    movel([0.601016, -1.382739, -2.575796, -0.753854, 1.570796, 2.171812],accel_mss,speed_ms,0,blend_radius_m)
    movel([0.599309, -1.384316, -2.574679, -0.753394, 1.570796, 2.170106],accel_mss,speed_ms,0,blend_radius_m)
    movel([0.597574, -1.385721, -2.573681, -0.752987, 1.570796, 2.168370],accel_mss,speed_ms,0,blend_radius_m)
    movel([0.595833, -1.386908, -2.572835, -0.752646, 1.570796, 2.166630],accel_mss,speed_ms,0,blend_radius_m)
    movel([0.594095, -1.387836, -2.572173, -0.752380, 1.570796, 2.164892],accel_mss,speed_ms,0,blend_radius_m)
    movel([0.592375, -1.388464, -2.571724, -0.752201, 1.570796, 2.163171],accel_mss,speed_ms,0,blend_radius_m)
    movel([0.590691, -1.388744, -2.571523, -0.752121, 1.570796, 2.161487],accel_mss,speed_ms,0,blend_radius_m)
    movel([0.589052, -1.388638, -2.571599, -0.752152, 1.570796, 2.159848],accel_mss,speed_ms,0,blend_radius_m)
    movel([0.588253, -1.388424, -2.571753, -0.752213, 1.570796, 2.159050],accel_mss,speed_ms,0,blend_radius_m)
    movel([0.587471, -1.388096, -2.571987, -0.752306, 1.570796, 2.158268],accel_mss,speed_ms,0,blend_radius_m)
    movel([0.585965, -1.387077, -2.572715, -0.752597, 1.570796, 2.156761],accel_mss,speed_ms,0,blend_radius_m)
    movel([0.584424, -1.385537, -2.573812, -0.753040, 1.570796, 2.155220],accel_mss,speed_ms,0,blend_radius_m)
    movel([0.583153, -1.383849, -2.575010, -0.753530, 1.570796, 2.153949],accel_mss,speed_ms,0,blend_radius_m)
    movel([0.582122, -1.382027, -2.576299, -0.754063, 1.570796, 2.152918],accel_mss,speed_ms,0,blend_radius_m)
    movel([0.581300, -1.380074, -2.577675, -0.754640, 1.570796, 2.152096],accel_mss,speed_ms,0,blend_radius_m)
    movel([0.580659, -1.378000, -2.579131, -0.755258, 1.570796, 2.151455],accel_mss,speed_ms,0,blend_radius_m)
    movel([0.580165, -1.375815, -2.580658, -0.755917, 1.570796, 2.150961],accel_mss,speed_ms,0,blend_radius_m)
    movel([0.579497, -1.371134, -2.583905, -0.757350, 1.570796, 2.150294],accel_mss,speed_ms,0,blend_radius_m)
    movel([0.578951, -1.365850, -2.587534, -0.759005, 1.570796, 2.149747],accel_mss,speed_ms,0,blend_radius_m)
    movel([0.578551, -1.360508, -2.591161, -0.760719, 1.570796, 2.149347],accel_mss,speed_ms,0,blend_radius_m)
    movel([0.578456, -1.355007, -2.594855, -0.762526, 1.570796, 2.149252],accel_mss,speed_ms,0,blend_radius_m)
    movel([0.578578, -1.352162, -2.596749, -0.763478, 1.570796, 2.149375],accel_mss,speed_ms,0,blend_radius_m)
    movel([0.578843, -1.349233, -2.598687, -0.764469, 1.570796, 2.149640],accel_mss,speed_ms,0,blend_radius_m)
    movel([0.579128, -1.345588, -2.601082, -0.765719, 1.570796, 2.149924],accel_mss,speed_ms,0,blend_radius_m)
    movel([0.579166, -1.341949, -2.603455, -0.766985, 1.570796, 2.149962],accel_mss,speed_ms,0,blend_radius_m)
    movel([0.578983, -1.338332, -2.605795, -0.768262, 1.570796, 2.149780],accel_mss,speed_ms,0,blend_radius_m)
    movel([0.578620, -1.334746, -2.608097, -0.769545, 1.570796, 2.149417],accel_mss,speed_ms,0,blend_radius_m)
    movel([0.577474, -1.327732, -2.612550, -0.772107, 1.570796, 2.148271],accel_mss,speed_ms,0,blend_radius_m)
    movel([0.576003, -1.321005, -2.616758, -0.774626, 1.570796, 2.146800],accel_mss,speed_ms,0,blend_radius_m)
    movel([0.574612, -1.316084, -2.619798, -0.776507, 1.570796, 2.145408],accel_mss,speed_ms,0,blend_radius_m)
    movel([0.572792, -1.311386, -2.622670, -0.778332, 1.570796, 2.143588],accel_mss,speed_ms,0,blend_radius_m)
    movel([0.570532, -1.306949, -2.625357, -0.780084, 1.570796, 2.141328],accel_mss,speed_ms,0,blend_radius_m)
    movel([0.567821, -1.302820, -2.627833, -0.781736, 1.570796, 2.138617],accel_mss,speed_ms,0,blend_radius_m)
    movel([0.564652, -1.299032, -2.630085, -0.783272, 1.570796, 2.135448],accel_mss,speed_ms,0,blend_radius_m)
    movel([0.562893, -1.297282, -2.631119, -0.783988, 1.570796, 2.133689],accel_mss,speed_ms,0,blend_radius_m)
    movel([0.559022, -1.294091, -2.632994, -0.785303, 1.570796, 2.129818],accel_mss,speed_ms,0,blend_radius_m)
    movel([0.556907, -1.292661, -2.633831, -0.785897, 1.570796, 2.127704],accel_mss,speed_ms,0,blend_radius_m)
    movel([0.552322, -1.290161, -2.635286, -0.786941, 1.570796, 2.123118],accel_mss,speed_ms,0,blend_radius_m)
    movel([0.548890, -1.288814, -2.636068, -0.787508, 1.570796, 2.119686],accel_mss,speed_ms,0,blend_radius_m)
    movel([0.545173, -1.287852, -2.636624, -0.787913, 1.570796, 2.115969],accel_mss,speed_ms,0,blend_radius_m)
    movel([0.541202, -1.287290, -2.636948, -0.788150, 1.570796, 2.111998],accel_mss,speed_ms,0,blend_radius_m)
    movel([0.537005, -1.287149, -2.637030, -0.788210, 1.570796, 2.107801],accel_mss,speed_ms,0,blend_radius_m)
    movel([0.532609, -1.287443, -2.636860, -0.788086, 1.570796, 2.103406],accel_mss,speed_ms,0,blend_radius_m)
    movel([0.528049, -1.288183, -2.636433, -0.787773, 1.570796, 2.098845],accel_mss,speed_ms,0,blend_radius_m)
    movel([0.523356, -1.289383, -2.635738, -0.787268, 1.570796, 2.094152],accel_mss,speed_ms,0,blend_radius_m)
    movel([0.518564, -1.291050, -2.634770, -0.786569, 1.570796, 2.089360],accel_mss,speed_ms,0,blend_radius_m)
    movel([0.514066, -1.292974, -2.633648, -0.785767, 1.570796, 2.084862],accel_mss,speed_ms,0,blend_radius_m)
    movel([0.509727, -1.295149, -2.632374, -0.784866, 1.570796, 2.080523],accel_mss,speed_ms,0,blend_radius_m)
    movel([0.505563, -1.297588, -2.630938, -0.783862, 1.570796, 2.076360],accel_mss,speed_ms,0,blend_radius_m)
    movel([0.501589, -1.300304, -2.629331, -0.782754, 1.570796, 2.072386],accel_mss,speed_ms,0,blend_radius_m)
    movel([0.499677, -1.301770, -2.628459, -0.782160, 1.570796, 2.070473],accel_mss,speed_ms,0,blend_radius_m)
    movel([0.496018, -1.304922, -2.626575, -0.780892, 1.570796, 2.066815],accel_mss,speed_ms,0,blend_radius_m)
    movel([0.494274, -1.306613, -2.625559, -0.780217, 1.570796, 2.065071],accel_mss,speed_ms,0,blend_radius_m)
    movel([0.490969, -1.310226, -2.623376, -0.778788, 1.570796, 2.061765],accel_mss,speed_ms,0,blend_radius_m)
    movel([0.489409, -1.312153, -2.622204, -0.778032, 1.570796, 2.060205],accel_mss,speed_ms,0,blend_radius_m)
    movel([0.487917, -1.314158, -2.620980, -0.777252, 1.570796, 2.058713],accel_mss,speed_ms,0,blend_radius_m)
    movel([0.485915, -1.317093, -2.619178, -0.776118, 1.570796, 2.056711],accel_mss,speed_ms,0,blend_radius_m)
    movel([0.484053, -1.320085, -2.617329, -0.774975, 1.570796, 2.054849],accel_mss,speed_ms,0,blend_radius_m)
    movel([0.482333, -1.323108, -2.615449, -0.773832, 1.570796, 2.053129],accel_mss,speed_ms,0,blend_radius_m)
    movel([0.480751, -1.326147, -2.613547, -0.772695, 1.570796, 2.051547],accel_mss,speed_ms,0,blend_radius_m)
    movel([0.479315, -1.329177, -2.611638, -0.771574, 1.570796, 2.050111],accel_mss,speed_ms,0,blend_radius_m)
    movel([0.478026, -1.332177, -2.609736, -0.770476, 1.570796, 2.048823],accel_mss,speed_ms,0,blend_radius_m)
    movel([0.476884, -1.335130, -2.607852, -0.769407, 1.570796, 2.047680],accel_mss,speed_ms,0,blend_radius_m)
    movel([0.475891, -1.338015, -2.605999, -0.768375, 1.570796, 2.046688],accel_mss,speed_ms,0,blend_radius_m)
    movel([0.472966, -1.349149, -2.598742, -0.764497, 1.570796, 2.043762],accel_mss,speed_ms,0,blend_radius_m)
    movel([0.470619, -1.357979, -2.592865, -0.761545, 1.570796, 2.041416],accel_mss,speed_ms,0,blend_radius_m)
    movel([0.470325, -1.358818, -2.592301, -0.761270, 1.570796, 2.041122],accel_mss,speed_ms,0,blend_radius_m)
    movel([0.475631, -1.356833, -2.593634, -0.761922, 1.570796, 2.046427],accel_mss,speed_ms,0,blend_radius_m)
    movel([0.480943, -1.355196, -2.594729, -0.762464, 1.570796, 2.051739],accel_mss,speed_ms,0,blend_radius_m)
    movel([0.486236, -1.353899, -2.595594, -0.762896, 1.570796, 2.057033],accel_mss,speed_ms,0,blend_radius_m)
    movel([0.491479, -1.352929, -2.596240, -0.763220, 1.570796, 2.062275],accel_mss,speed_ms,0,blend_radius_m)
    movel([0.496639, -1.352279, -2.596672, -0.763438, 1.570796, 2.067435],accel_mss,speed_ms,0,blend_radius_m)
    movel([0.501690, -1.351932, -2.596902, -0.763555, 1.570796, 2.072486],accel_mss,speed_ms,0,blend_radius_m)
    movel([0.506601, -1.351881, -2.596936, -0.763573, 1.570796, 2.077398],accel_mss,speed_ms,0,blend_radius_m)
    movel([0.511345, -1.352106, -2.596786, -0.763497, 1.570796, 2.082141],accel_mss,speed_ms,0,blend_radius_m)
    movel([0.513503, -1.352345, -2.596628, -0.763416, 1.570796, 2.084300],accel_mss,speed_ms,0,blend_radius_m)
    movel([0.515622, -1.352729, -2.596373, -0.763287, 1.570796, 2.086418],accel_mss,speed_ms,0,blend_radius_m)
    movel([0.517679, -1.353257, -2.596022, -0.763110, 1.570796, 2.088475],accel_mss,speed_ms,0,blend_radius_m)
    movel([0.519651, -1.353929, -2.595574, -0.762885, 1.570796, 2.090447],accel_mss,speed_ms,0,blend_radius_m)
    movel([0.521517, -1.354747, -2.595029, -0.762613, 1.570796, 2.092314],accel_mss,speed_ms,0,blend_radius_m)
    movel([0.523257, -1.355711, -2.594385, -0.762293, 1.570796, 2.094053],accel_mss,speed_ms,0,blend_radius_m)
    movel([0.524849, -1.356818, -2.593644, -0.761927, 1.570796, 2.095645],accel_mss,speed_ms,0,blend_radius_m)
    movel([0.526273, -1.358067, -2.592806, -0.761516, 1.570796, 2.097069],accel_mss,speed_ms,0,blend_radius_m)
    movel([0.527508, -1.359460, -2.591868, -0.761060, 1.570796, 2.098304],accel_mss,speed_ms,0,blend_radius_m)
    movel([0.528536, -1.360996, -2.590832, -0.760561, 1.570796, 2.099332],accel_mss,speed_ms,0,blend_radius_m)
    movel([0.529334, -1.362671, -2.589697, -0.760020, 1.570796, 2.100130],accel_mss,speed_ms,0,blend_radius_m)
    movel([0.529883, -1.364486, -2.588464, -0.759439, 1.570796, 2.100680],accel_mss,speed_ms,0,blend_radius_m)
    movel([0.530165, -1.366437, -2.587133, -0.758820, 1.570796, 2.100962],accel_mss,speed_ms,0,blend_radius_m)
    movel([0.530163, -1.368526, -2.585701, -0.758162, 1.570796, 2.100960],accel_mss,speed_ms,0,blend_radius_m)
    movel([0.529857, -1.370747, -2.584172, -0.757470, 1.570796, 2.100654],accel_mss,speed_ms,0,blend_radius_m)
    movel([0.529228, -1.373102, -2.582544, -0.756743, 1.570796, 2.100024],accel_mss,speed_ms,0,blend_radius_m)
    movel([0.528005, -1.376258, -2.580348, -0.755782, 1.570796, 2.098801],accel_mss,speed_ms,0,blend_radius_m)
    movel([0.526428, -1.379471, -2.578099, -0.754819, 1.570796, 2.097224],accel_mss,speed_ms,0,blend_radius_m)
    movel([0.524564, -1.382702, -2.575822, -0.753865, 1.570796, 2.095360],accel_mss,speed_ms,0,blend_radius_m)
    movel([0.522477, -1.385922, -2.573537, -0.752929, 1.570796, 2.093273],accel_mss,speed_ms,0,blend_radius_m)
    movel([0.520232, -1.389098, -2.571270, -0.752021, 1.570796, 2.091028],accel_mss,speed_ms,0,blend_radius_m)
    movel([0.517887, -1.392198, -2.569042, -0.751149, 1.570796, 2.088683],accel_mss,speed_ms,0,blend_radius_m)
    movel([0.513159, -1.398048, -2.564800, -0.749541, 1.570796, 2.083955],accel_mss,speed_ms,0,blend_radius_m)
    movel([0.510054, -1.401623, -2.562183, -0.748583, 1.570796, 2.080850],accel_mss,speed_ms,0,blend_radius_m)
    movel([0.506857, -1.405036, -2.559666, -0.747687, 1.570796, 2.077653],accel_mss,speed_ms,0,blend_radius_m)
    movel([0.503577, -1.408310, -2.557236, -0.746843, 1.570796, 2.074373],accel_mss,speed_ms,0,blend_radius_m)
    movel([0.500217, -1.411476, -2.554871, -0.746042, 1.570796, 2.071013],accel_mss,speed_ms,0,blend_radius_m)
    movel([0.496786, -1.414553, -2.552558, -0.745278, 1.570796, 2.067583],accel_mss,speed_ms,0,blend_radius_m)
    movel([0.493292, -1.417568, -2.550278, -0.744543, 1.570796, 2.064088],accel_mss,speed_ms,0,blend_radius_m)
    movel([0.486129, -1.423508, -2.545746, -0.743135, 1.570796, 2.056925],accel_mss,speed_ms,0,blend_radius_m)
    movel([0.487951, -1.426525, -2.543424, -0.742440, 1.570796, 2.058747],accel_mss,speed_ms,0,blend_radius_m)
    movel([0.488812, -1.428211, -2.542120, -0.742058, 1.570796, 2.059609],accel_mss,speed_ms,0,blend_radius_m)
    movel([0.489370, -1.429952, -2.540769, -0.741667, 1.570796, 2.060166],accel_mss,speed_ms,0,blend_radius_m)
    movel([0.489470, -1.430830, -2.540087, -0.741472, 1.570796, 2.060266],accel_mss,speed_ms,0,blend_radius_m)
    movel([0.489417, -1.431705, -2.539405, -0.741279, 1.570796, 2.060213],accel_mss,speed_ms,0,blend_radius_m)
    movel([0.489187, -1.432571, -2.538729, -0.741089, 1.570796, 2.059983],accel_mss,speed_ms,0,blend_radius_m)
    movel([0.488755, -1.433422, -2.538064, -0.740904, 1.570796, 2.059551],accel_mss,speed_ms,0,blend_radius_m)
    movel([0.488098, -1.434250, -2.537415, -0.740724, 1.570796, 2.058895],accel_mss,speed_ms,0,blend_radius_m)
    movel([0.487186, -1.435055, -2.536784, -0.740550, 1.570796, 2.057983],accel_mss,speed_ms,0,blend_radius_m)
    movel([0.485997, -1.435830, -2.536175, -0.740384, 1.570796, 2.056793],accel_mss,speed_ms,0,blend_radius_m)
    movel([0.484506, -1.436568, -2.535594, -0.740227, 1.570796, 2.055302],accel_mss,speed_ms,0,blend_radius_m)
    movel([0.483220, -1.437075, -2.535195, -0.740119, 1.570796, 2.054016],accel_mss,speed_ms,0,blend_radius_m)
    movel([0.482001, -1.437448, -2.534901, -0.740040, 1.570796, 2.052798],accel_mss,speed_ms,0,blend_radius_m)
    movel([0.480845, -1.437700, -2.534702, -0.739987, 1.570796, 2.051642],accel_mss,speed_ms,0,blend_radius_m)
    movel([0.478697, -1.437878, -2.534562, -0.739949, 1.570796, 2.049493],accel_mss,speed_ms,0,blend_radius_m)
    movel([0.477695, -1.437824, -2.534604, -0.739961, 1.570796, 2.048491],accel_mss,speed_ms,0,blend_radius_m)
    movel([0.475806, -1.437485, -2.534871, -0.740032, 1.570796, 2.046602],accel_mss,speed_ms,0,blend_radius_m)
    movel([0.474040, -1.436905, -2.535329, -0.740155, 1.570796, 2.044837],accel_mss,speed_ms,0,blend_radius_m)
    movel([0.472356, -1.436162, -2.535914, -0.740313, 1.570796, 2.043153],accel_mss,speed_ms,0,blend_radius_m)
    movel([0.469076, -1.434521, -2.537203, -0.740665, 1.570796, 2.039872],accel_mss,speed_ms,0,blend_radius_m)
    movel([0.465722, -1.436483, -2.535661, -0.740245, 1.570796, 2.036518],accel_mss,speed_ms,0,blend_radius_m)
    movel([0.463980, -1.437385, -2.534950, -0.740053, 1.570796, 2.034776],accel_mss,speed_ms,0,blend_radius_m)
    movel([0.462220, -1.438181, -2.534322, -0.739885, 1.570796, 2.033016],accel_mss,speed_ms,0,blend_radius_m)
    movel([0.460464, -1.438828, -2.533812, -0.739750, 1.570796, 2.031260],accel_mss,speed_ms,0,blend_radius_m)
    movel([0.458733, -1.439284, -2.533451, -0.739654, 1.570796, 2.029530],accel_mss,speed_ms,0,blend_radius_m)
    movel([0.457049, -1.439507, -2.533274, -0.739608, 1.570796, 2.027846],accel_mss,speed_ms,0,blend_radius_m)
    movel([0.455428, -1.439456, -2.533315, -0.739619, 1.570796, 2.026225],accel_mss,speed_ms,0,blend_radius_m)
    movel([0.454430, -1.439177, -2.533536, -0.739677, 1.570796, 2.025226],accel_mss,speed_ms,0,blend_radius_m)
    movel([0.453802, -1.438678, -2.533930, -0.739781, 1.570796, 2.024598],accel_mss,speed_ms,0,blend_radius_m)
    movel([0.453497, -1.437998, -2.534467, -0.739924, 1.570796, 2.024293],accel_mss,speed_ms,0,blend_radius_m)
    movel([0.453470, -1.437176, -2.535115, -0.740098, 1.570796, 2.024266],accel_mss,speed_ms,0,blend_radius_m)
    movel([0.453674, -1.436249, -2.535845, -0.740295, 1.570796, 2.024470],accel_mss,speed_ms,0,blend_radius_m)
    movel([0.454060, -1.435263, -2.536620, -0.740506, 1.570796, 2.024857],accel_mss,speed_ms,0,blend_radius_m)
    movel([0.454581, -1.434254, -2.537412, -0.740723, 1.570796, 2.025378],accel_mss,speed_ms,0,blend_radius_m)
    movel([0.455194, -1.433264, -2.538187, -0.740938, 1.570796, 2.025991],accel_mss,speed_ms,0,blend_radius_m)
    movel([0.456666, -1.431232, -2.539773, -0.741384, 1.570796, 2.027463],accel_mss,speed_ms,0,blend_radius_m)
    movel([0.458291, -1.429284, -2.541288, -0.741817, 1.570796, 2.029088],accel_mss,speed_ms,0,blend_radius_m)
    movel([0.461810, -1.425442, -2.544259, -0.742688, 1.570796, 2.032606],accel_mss,speed_ms,0,blend_radius_m)
    movel([0.459726, -1.420705, -2.547891, -0.743793, 1.570796, 2.030522],accel_mss,speed_ms,0,blend_radius_m)
    movel([0.457477, -1.416035, -2.551439, -0.744915, 1.570796, 2.028274],accel_mss,speed_ms,0,blend_radius_m)
    movel([0.455278, -1.411296, -2.555006, -0.746087, 1.570796, 2.026074],accel_mss,speed_ms,0,blend_radius_m)
    movel([0.454264, -1.408857, -2.556829, -0.746703, 1.570796, 2.025061],accel_mss,speed_ms,0,blend_radius_m)
    movel([0.453345, -1.406346, -2.558696, -0.747347, 1.570796, 2.024141],accel_mss,speed_ms,0,blend_radius_m)
    movel([0.452586, -1.403861, -2.560535, -0.747994, 1.570796, 2.023383],accel_mss,speed_ms,0,blend_radius_m)
    movel([0.451946, -1.401323, -2.562403, -0.748663, 1.570796, 2.022742],accel_mss,speed_ms,0,blend_radius_m)
    movel([0.450899, -1.396130, -2.566196, -0.750063, 1.570796, 2.021696],accel_mss,speed_ms,0,blend_radius_m)
    movel([0.449938, -1.390874, -2.569995, -0.751519, 1.570796, 2.020735],accel_mss,speed_ms,0,blend_radius_m)
    movel([0.448799, -1.385666, -2.573720, -0.753003, 1.570796, 2.019595],accel_mss,speed_ms,0,blend_radius_m)
    movel([0.446490, -1.387724, -2.572253, -0.752412, 1.570796, 2.017286],accel_mss,speed_ms,0,blend_radius_m)
    movel([0.444290, -1.389839, -2.570739, -0.751811, 1.570796, 2.015086],accel_mss,speed_ms,0,blend_radius_m)
    movel([0.442204, -1.392001, -2.569185, -0.751204, 1.570796, 2.013001],accel_mss,speed_ms,0,blend_radius_m)
    movel([0.440236, -1.394203, -2.567594, -0.750592, 1.570796, 2.011032],accel_mss,speed_ms,0,blend_radius_m)
    movel([0.438387, -1.396442, -2.565970, -0.749978, 1.570796, 2.009184],accel_mss,speed_ms,0,blend_radius_m)
    movel([0.436661, -1.398709, -2.564318, -0.749363, 1.570796, 2.007457],accel_mss,speed_ms,0,blend_radius_m)
    movel([0.435061, -1.401000, -2.562640, -0.748749, 1.570796, 2.005857],accel_mss,speed_ms,0,blend_radius_m)
    movel([0.433585, -1.403309, -2.560941, -0.748138, 1.570796, 2.004382],accel_mss,speed_ms,0,blend_radius_m)
    movel([0.432240, -1.405632, -2.559225, -0.747532, 1.570796, 2.003037],accel_mss,speed_ms,0,blend_radius_m)
    movel([0.431031, -1.407960, -2.557497, -0.746932, 1.570796, 2.001827],accel_mss,speed_ms,0,blend_radius_m)
    movel([0.429952, -1.410292, -2.555757, -0.746340, 1.570796, 2.000748],accel_mss,speed_ms,0,blend_radius_m)
    movel([0.429009, -1.412619, -2.554014, -0.745756, 1.570796, 1.999805],accel_mss,speed_ms,0,blend_radius_m)
    movel([0.428208, -1.414937, -2.552269, -0.745184, 1.570796, 1.999004],accel_mss,speed_ms,0,blend_radius_m)
    movel([0.427544, -1.417243, -2.550524, -0.744621, 1.570796, 1.998340],accel_mss,speed_ms,0,blend_radius_m)
    movel([0.427022, -1.419531, -2.548787, -0.744072, 1.570796, 1.997819],accel_mss,speed_ms,0,blend_radius_m)
    movel([0.426645, -1.421797, -2.547057, -0.743535, 1.570796, 1.997441],accel_mss,speed_ms,0,blend_radius_m)
    movel([0.426336, -1.425233, -2.544420, -0.742736, 1.570796, 1.997132],accel_mss,speed_ms,0,blend_radius_m)
    movel([0.426338, -1.428536, -2.541869, -0.741985, 1.570796, 1.997134],accel_mss,speed_ms,0,blend_radius_m)
    movel([0.426615, -1.431713, -2.539399, -0.741278, 1.570796, 1.997412],accel_mss,speed_ms,0,blend_radius_m)
    movel([0.427143, -1.434772, -2.537005, -0.740611, 1.570796, 1.997939],accel_mss,speed_ms,0,blend_radius_m)
    movel([0.427888, -1.437723, -2.534684, -0.739982, 1.570796, 1.998684],accel_mss,speed_ms,0,blend_radius_m)
    movel([0.428821, -1.440571, -2.532431, -0.739387, 1.570796, 1.999617],accel_mss,speed_ms,0,blend_radius_m)
    movel([0.429912, -1.443324, -2.530241, -0.738824, 1.570796, 2.000708],accel_mss,speed_ms,0,blend_radius_m)
    movel([0.431139, -1.445987, -2.528112, -0.738291, 1.570796, 2.001935],accel_mss,speed_ms,0,blend_radius_m)
    movel([0.433874, -1.451135, -2.523964, -0.737290, 1.570796, 2.004670],accel_mss,speed_ms,0,blend_radius_m)
    movel([0.436780, -1.456133, -2.519898, -0.736358, 1.570796, 2.007576],accel_mss,speed_ms,0,blend_radius_m)
    movel([0.438913, -1.460048, -2.516686, -0.735654, 1.570796, 2.009709],accel_mss,speed_ms,0,blend_radius_m)
    movel([0.439725, -1.461265, -2.515683, -0.735441, 1.570796, 2.010521],accel_mss,speed_ms,0,blend_radius_m)
    movel([0.441334, -1.463212, -2.514074, -0.735104, 1.570796, 2.012131],accel_mss,speed_ms,0,blend_radius_m)
    movel([0.441603, -1.463733, -2.513641, -0.735014, 1.570796, 2.012400],accel_mss,speed_ms,0,blend_radius_m)
    movel([0.441772, -1.464329, -2.513148, -0.734913, 1.570796, 2.012569],accel_mss,speed_ms,0,blend_radius_m)
    movel([0.441813, -1.465029, -2.512566, -0.734794, 1.570796, 2.012609],accel_mss,speed_ms,0,blend_radius_m)
    movel([0.441699, -1.465863, -2.511872, -0.734654, 1.570796, 2.012495],accel_mss,speed_ms,0,blend_radius_m)
    movel([0.441396, -1.466857, -2.511044, -0.734488, 1.570796, 2.012192],accel_mss,speed_ms,0,blend_radius_m)
    movel([0.440931, -1.467831, -2.510231, -0.734327, 1.570796, 2.011727],accel_mss,speed_ms,0,blend_radius_m)
    movel([0.440325, -1.468778, -2.509438, -0.734172, 1.570796, 2.011121],accel_mss,speed_ms,0,blend_radius_m)
    movel([0.439590, -1.469700, -2.508666, -0.734023, 1.570796, 2.010386],accel_mss,speed_ms,0,blend_radius_m)
    movel([0.438746, -1.470588, -2.507921, -0.733880, 1.570796, 2.009543],accel_mss,speed_ms,0,blend_radius_m)
    movel([0.436787, -1.472256, -2.506518, -0.733615, 1.570796, 2.007583],accel_mss,speed_ms,0,blend_radius_m)
    movel([0.435704, -1.473027, -2.505868, -0.733494, 1.570796, 2.006500],accel_mss,speed_ms,0,blend_radius_m)
    movel([0.433416, -1.474430, -2.504683, -0.733276, 1.570796, 2.004212],accel_mss,speed_ms,0,blend_radius_m)
    movel([0.431061, -1.475618, -2.503677, -0.733094, 1.570796, 2.001858],accel_mss,speed_ms,0,blend_radius_m)
    movel([0.428771, -1.476565, -2.502874, -0.732951, 1.570796, 1.999567],accel_mss,speed_ms,0,blend_radius_m)
    movel([0.426663, -1.477239, -2.502301, -0.732849, 1.570796, 1.997460],accel_mss,speed_ms,0,blend_radius_m)
    movel([0.423583, -1.477897, -2.501741, -0.732751, 1.570796, 1.994379],accel_mss,speed_ms,0,blend_radius_m)
    movel([0.422062, -1.478099, -2.501569, -0.732721, 1.570796, 1.992858],accel_mss,speed_ms,0,blend_radius_m)
    movel([0.420564, -1.478215, -2.501470, -0.732704, 1.570796, 1.991361],accel_mss,speed_ms,0,blend_radius_m)
    movel([0.417652, -1.478202, -2.501481, -0.732706, 1.570796, 1.988449],accel_mss,speed_ms,0,blend_radius_m)
    movel([0.414889, -1.477867, -2.501766, -0.732755, 1.570796, 1.985685],accel_mss,speed_ms,0,blend_radius_m)
    movel([0.412317, -1.477216, -2.502320, -0.732853, 1.570796, 1.983113],accel_mss,speed_ms,0,blend_radius_m)
    movel([0.409984, -1.476259, -2.503133, -0.732997, 1.570796, 1.980780],accel_mss,speed_ms,0,blend_radius_m)
    movel([0.408920, -1.475665, -2.503637, -0.733087, 1.570796, 1.979717],accel_mss,speed_ms,0,blend_radius_m)
    movel([0.407027, -1.474254, -2.504832, -0.733303, 1.570796, 1.977823],accel_mss,speed_ms,0,blend_radius_m)
    movel([0.406209, -1.473436, -2.505523, -0.733430, 1.570796, 1.977005],accel_mss,speed_ms,0,blend_radius_m)
    movel([0.405259, -1.472249, -2.506525, -0.733616, 1.570796, 1.976055],accel_mss,speed_ms,0,blend_radius_m)
    movel([0.404449, -1.470964, -2.507605, -0.733820, 1.570796, 1.975245],accel_mss,speed_ms,0,blend_radius_m)
    movel([0.403764, -1.469596, -2.508754, -0.734039, 1.570796, 1.974560],accel_mss,speed_ms,0,blend_radius_m)
    movel([0.403183, -1.468158, -2.509957, -0.734274, 1.570796, 1.973979],accel_mss,speed_ms,0,blend_radius_m)
    movel([0.402266, -1.465126, -2.512485, -0.734778, 1.570796, 1.973062],accel_mss,speed_ms,0,blend_radius_m)
    movel([0.401556, -1.461978, -2.515095, -0.735317, 1.570796, 1.972352],accel_mss,speed_ms,0,blend_radius_m)
    movel([0.400830, -1.457941, -2.518418, -0.736030, 1.570796, 1.971627],accel_mss,speed_ms,0,blend_radius_m)
    movel([0.400308, -1.453769, -2.521826, -0.736794, 1.570796, 1.971104],accel_mss,speed_ms,0,blend_radius_m)
    movel([0.400013, -1.449467, -2.525313, -0.737610, 1.570796, 1.970809],accel_mss,speed_ms,0,blend_radius_m)
    movel([0.399967, -1.445042, -2.528868, -0.738479, 1.570796, 1.970763],accel_mss,speed_ms,0,blend_radius_m)
    movel([0.400195, -1.440500, -2.532487, -0.739402, 1.570796, 1.970991],accel_mss,speed_ms,0,blend_radius_m)
    movel([0.400723, -1.435849, -2.536160, -0.740380, 1.570796, 1.971519],accel_mss,speed_ms,0,blend_radius_m)
    movel([0.401573, -1.431098, -2.539878, -0.741413, 1.570796, 1.972369],accel_mss,speed_ms,0,blend_radius_m)
    movel([0.402770, -1.426254, -2.543633, -0.742502, 1.570796, 1.973566],accel_mss,speed_ms,0,blend_radius_m)
    movel([0.403900, -1.422554, -2.546477, -0.743357, 1.570796, 1.974696],accel_mss,speed_ms,0,blend_radius_m)
    movel([0.405261, -1.418682, -2.549432, -0.744275, 1.570796, 1.976057],accel_mss,speed_ms,0,blend_radius_m)
    movel([0.406863, -1.414688, -2.552457, -0.745245, 1.570796, 1.977659],accel_mss,speed_ms,0,blend_radius_m)
    movel([0.408709, -1.410630, -2.555504, -0.746254, 1.570796, 1.979506],accel_mss,speed_ms,0,blend_radius_m)
    movel([0.410809, -1.406568, -2.558531, -0.747290, 1.570796, 1.981605],accel_mss,speed_ms,0,blend_radius_m)
    movel([0.413166, -1.402564, -2.561491, -0.748335, 1.570796, 1.983963],accel_mss,speed_ms,0,blend_radius_m)
    movel([0.415786, -1.398674, -2.564343, -0.749372, 1.570796, 1.986582],accel_mss,speed_ms,0,blend_radius_m)
    movel([0.417196, -1.396792, -2.565715, -0.749882, 1.570796, 1.987993],accel_mss,speed_ms,0,blend_radius_m)
    movel([0.418672, -1.394964, -2.567042, -0.750382, 1.570796, 1.989469],accel_mss,speed_ms,0,blend_radius_m)
    movel([0.421615, -1.391625, -2.569455, -0.751309, 1.570796, 1.992411],accel_mss,speed_ms,0,blend_radius_m)
    movel([0.424754, -1.388374, -2.571788, -0.752227, 1.570796, 1.995550],accel_mss,speed_ms,0,blend_radius_m)
    movel([0.428078, -1.385228, -2.574031, -0.753130, 1.570796, 1.998875],accel_mss,speed_ms,0,blend_radius_m)
    movel([0.431568, -1.382200, -2.576177, -0.754012, 1.570796, 2.002364],accel_mss,speed_ms,0,blend_radius_m)
    movel([0.435213, -1.379311, -2.578212, -0.754867, 1.570796, 2.006009],accel_mss,speed_ms,0,blend_radius_m)
    movel([0.438991, -1.376573, -2.580129, -0.755687, 1.570796, 2.009787],accel_mss,speed_ms,0,blend_radius_m)
    movel([0.442888, -1.374005, -2.581917, -0.756467, 1.570796, 2.013684],accel_mss,speed_ms,0,blend_radius_m)
    movel([0.446886, -1.371627, -2.583565, -0.757197, 1.570796, 2.017683],accel_mss,speed_ms,0,blend_radius_m)
    movel([0.447752, -1.362373, -2.589900, -0.760117, 1.570796, 2.018549],accel_mss,speed_ms,0,blend_radius_m)
    movel([0.448207, -1.357694, -2.593056, -0.761638, 1.570796, 2.019003],accel_mss,speed_ms,0,blend_radius_m)
    movel([0.448864, -1.352921, -2.596245, -0.763223, 1.570796, 2.019660],accel_mss,speed_ms,0,blend_radius_m)
    movel([0.449625, -1.349269, -2.598663, -0.764457, 1.570796, 2.020421],accel_mss,speed_ms,0,blend_radius_m)
    movel([0.450699, -1.345531, -2.601119, -0.765739, 1.570796, 2.021496],accel_mss,speed_ms,0,blend_radius_m)
    movel([0.452068, -1.341722, -2.603602, -0.767065, 1.570796, 2.022864],accel_mss,speed_ms,0,blend_radius_m)
    movel([0.453719, -1.337851, -2.606104, -0.768433, 1.570796, 2.024516],accel_mss,speed_ms,0,blend_radius_m)
    movel([0.455637, -1.333936, -2.608615, -0.769838, 1.570796, 2.026434],accel_mss,speed_ms,0,blend_radius_m)
    movel([0.457808, -1.329990, -2.611124, -0.771275, 1.570796, 2.028604],accel_mss,speed_ms,0,blend_radius_m)
    movel([0.460215, -1.326025, -2.613624, -0.772740, 1.570796, 2.031012],accel_mss,speed_ms,0,blend_radius_m)
    movel([0.462843, -1.322058, -2.616103, -0.774227, 1.570796, 2.033639],accel_mss,speed_ms,0,blend_radius_m)
    movel([0.465673, -1.318108, -2.618552, -0.775729, 1.570796, 2.036469],accel_mss,speed_ms,0,blend_radius_m)
    movel([0.468693, -1.314186, -2.620962, -0.777241, 1.570796, 2.039490],accel_mss,speed_ms,0,blend_radius_m)
    movel([0.471884, -1.310311, -2.623324, -0.778754, 1.570796, 2.042681],accel_mss,speed_ms,0,blend_radius_m)
    movel([0.475227, -1.306500, -2.625627, -0.780262, 1.570796, 2.046023],accel_mss,speed_ms,0,blend_radius_m)
    movel([0.478703, -1.302770, -2.627863, -0.781756, 1.570796, 2.049500],accel_mss,speed_ms,0,blend_radius_m)
    movel([0.482290, -1.299142, -2.630020, -0.783227, 1.570796, 2.053086],accel_mss,speed_ms,0,blend_radius_m)
    movel([0.485975, -1.295631, -2.632091, -0.784667, 1.570796, 2.056771],accel_mss,speed_ms,0,blend_radius_m)
    movel([0.489731, -1.292257, -2.634067, -0.786065, 1.570796, 2.060527],accel_mss,speed_ms,0,blend_radius_m)
    movel([0.496968, -1.286144, -2.637609, -0.788636, 1.570796, 2.067764],accel_mss,speed_ms,0,blend_radius_m)
    movel([0.500705, -1.283179, -2.639309, -0.789900, 1.570796, 2.071501],accel_mss,speed_ms,0,blend_radius_m)
    movel([0.504524, -1.280314, -2.640943, -0.791132, 1.570796, 2.075320],accel_mss,speed_ms,0,blend_radius_m)
    movel([0.508425, -1.277585, -2.642488, -0.792315, 1.570796, 2.079222],accel_mss,speed_ms,0,blend_radius_m)
    movel([0.512405, -1.275028, -2.643928, -0.793432, 1.570796, 2.083201],accel_mss,speed_ms,0,blend_radius_m)
    movel([0.516463, -1.272675, -2.645246, -0.794468, 1.570796, 2.087259],accel_mss,speed_ms,0,blend_radius_m)
    movel([0.520598, -1.270562, -2.646424, -0.795403, 1.570796, 2.091394],accel_mss,speed_ms,0,blend_radius_m)
    movel([0.525247, -1.268505, -2.647565, -0.796319, 1.570796, 2.096043],accel_mss,speed_ms,0,blend_radius_m)
    movel([0.529924, -1.266727, -2.648547, -0.797115, 1.570796, 2.100720],accel_mss,speed_ms,0,blend_radius_m)
    movel([0.534608, -1.265225, -2.649373, -0.797791, 1.570796, 2.105404],accel_mss,speed_ms,0,blend_radius_m)
    movel([0.539277, -1.263999, -2.650046, -0.798344, 1.570796, 2.110073],accel_mss,speed_ms,0,blend_radius_m)
    movel([0.543909, -1.263050, -2.650565, -0.798774, 1.570796, 2.114705],accel_mss,speed_ms,0,blend_radius_m)
    movel([0.548480, -1.262375, -2.650934, -0.799080, 1.570796, 2.119276],accel_mss,speed_ms,0,blend_radius_m)
    movel([0.552974, -1.261971, -2.651155, -0.799264, 1.570796, 2.123770],accel_mss,speed_ms,0,blend_radius_m)
    movel([0.557365, -1.261835, -2.651229, -0.799326, 1.570796, 2.128162],accel_mss,speed_ms,0,blend_radius_m)
    movel([0.561634, -1.261965, -2.651158, -0.799266, 1.570796, 2.132430],accel_mss,speed_ms,0,blend_radius_m)
    movel([0.565759, -1.262351, -2.650947, -0.799091, 1.570796, 2.136556],accel_mss,speed_ms,0,blend_radius_m)
    movel([0.569723, -1.262993, -2.650596, -0.798799, 1.570796, 2.140519],accel_mss,speed_ms,0,blend_radius_m)
    movel([0.573505, -1.263882, -2.650110, -0.798397, 1.570796, 2.144301],accel_mss,speed_ms,0,blend_radius_m)
    movel([0.577085, -1.265010, -2.649491, -0.797888, 1.570796, 2.147881],accel_mss,speed_ms,0,blend_radius_m)
    movel([0.580448, -1.266370, -2.648743, -0.797275, 1.570796, 2.151244],accel_mss,speed_ms,0,blend_radius_m)
    movel([0.583576, -1.267954, -2.647869, -0.796565, 1.570796, 2.154372],accel_mss,speed_ms,0,blend_radius_m)
    movel([0.586452, -1.269757, -2.646871, -0.795761, 1.570796, 2.157249],accel_mss,speed_ms,0,blend_radius_m)
    movel([0.589310, -1.271851, -2.645706, -0.794832, 1.570796, 2.160106],accel_mss,speed_ms,0,blend_radius_m)
    movel([0.592005, -1.274099, -2.644449, -0.793840, 1.570796, 2.162801],accel_mss,speed_ms,0,blend_radius_m)
    movel([0.594490, -1.276534, -2.643081, -0.792774, 1.570796, 2.165286],accel_mss,speed_ms,0,blend_radius_m)
    movel([0.596713, -1.279192, -2.641579, -0.791618, 1.570796, 2.167509],accel_mss,speed_ms,0,blend_radius_m)
    movel([0.598939, -1.282605, -2.639638, -0.790146, 1.570796, 2.169736],accel_mss,speed_ms,0,blend_radius_m)
    movel([0.600795, -1.286342, -2.637495, -0.788552, 1.570796, 2.171591],accel_mss,speed_ms,0,blend_radius_m)
    movel([0.602271, -1.290357, -2.635173, -0.786859, 1.570796, 2.173068],accel_mss,speed_ms,0,blend_radius_m)
    movel([0.603362, -1.294601, -2.632696, -0.785092, 1.570796, 2.174158],accel_mss,speed_ms,0,blend_radius_m)
    movel([0.604062, -1.299028, -2.630087, -0.783274, 1.570796, 2.174858],accel_mss,speed_ms,0,blend_radius_m)
    movel([0.604367, -1.303592, -2.627371, -0.781425, 1.570796, 2.175163],accel_mss,speed_ms,0,blend_radius_m)
    movel([0.604275, -1.308247, -2.624573, -0.779569, 1.570796, 2.175072],accel_mss,speed_ms,0,blend_radius_m)
    movel([0.603783, -1.312952, -2.621716, -0.777720, 1.570796, 2.174579],accel_mss,speed_ms,0,blend_radius_m)
    movel([0.602354, -1.322280, -2.615965, -0.774143, 1.570796, 2.173150],accel_mss,speed_ms,0,blend_radius_m)
    movel([0.601466, -1.326921, -2.613061, -0.772407, 1.570796, 2.172262],accel_mss,speed_ms,0,blend_radius_m)
    movel([0.600320, -1.331659, -2.610065, -0.770665, 1.570796, 2.171117],accel_mss,speed_ms,0,blend_radius_m)
    movel([0.598313, -1.339603, -2.604975, -0.767811, 1.570796, 2.169110],accel_mss,speed_ms,0,blend_radius_m)
    movel([0.597505, -1.343557, -2.602409, -0.766424, 1.570796, 2.168301],accel_mss,speed_ms,0,blend_radius_m)
    movel([0.596910, -1.347433, -2.599872, -0.765084, 1.570796, 2.167707],accel_mss,speed_ms,0,blend_radius_m)
    movel([0.596598, -1.351193, -2.597392, -0.763804, 1.570796, 2.167394],accel_mss,speed_ms,0,blend_radius_m)
    movel([0.596623, -1.354787, -2.595002, -0.762600, 1.570796, 2.167420],accel_mss,speed_ms,0,blend_radius_m)
    movel([0.597053, -1.358178, -2.592732, -0.761480, 1.570796, 2.167849],accel_mss,speed_ms,0,blend_radius_m)
    movel([0.597944, -1.361320, -2.590613, -0.760456, 1.570796, 2.168740],accel_mss,speed_ms,0,blend_radius_m)
    movel([0.598482, -1.362473, -2.589832, -0.760084, 1.570796, 2.169278],accel_mss,speed_ms,0,blend_radius_m)
    movel([0.599238, -1.363462, -2.589160, -0.759767, 1.570796, 2.170034],accel_mss,speed_ms,0,blend_radius_m)
    movel([0.599719, -1.363846, -2.588899, -0.759644, 1.570796, 2.170515],accel_mss,speed_ms,0,blend_radius_m)
    movel([0.600276, -1.364131, -2.588706, -0.759553, 1.570796, 2.171072],accel_mss,speed_ms,0,blend_radius_m)
    movel([0.600918, -1.364298, -2.588592, -0.759499, 1.570796, 2.171715],accel_mss,speed_ms,0,blend_radius_m)
    movel([0.601653, -1.364323, -2.588575, -0.759491, 1.570796, 2.172450],accel_mss,speed_ms,0,blend_radius_m)
    movel([0.602474, -1.364194, -2.588663, -0.759532, 1.570796, 2.173270],accel_mss,speed_ms,0,blend_radius_m)
    movel([0.603319, -1.363925, -2.588846, -0.759618, 1.570796, 2.174116],accel_mss,speed_ms,0,blend_radius_m)
    movel([0.605012, -1.363089, -2.589414, -0.759886, 1.570796, 2.175808],accel_mss,speed_ms,0,blend_radius_m)
    movel([0.606146, -1.362357, -2.589911, -0.760122, 1.570796, 2.176942],accel_mss,speed_ms,0,blend_radius_m)
    movel([0.607218, -1.361544, -2.590461, -0.760384, 1.570796, 2.178014],accel_mss,speed_ms,0,blend_radius_m)
    movel([0.609185, -1.359710, -2.591700, -0.760979, 1.570796, 2.179982],accel_mss,speed_ms,0,blend_radius_m)
    movel([0.610927, -1.357656, -2.593082, -0.761651, 1.570796, 2.181724],accel_mss,speed_ms,0,blend_radius_m)
    movel([0.612463, -1.355446, -2.594562, -0.762381, 1.570796, 2.183260],accel_mss,speed_ms,0,blend_radius_m)
    movel([0.613804, -1.353151, -2.596092, -0.763146, 1.570796, 2.184600],accel_mss,speed_ms,0,blend_radius_m)
    movel([0.614965, -1.350838, -2.597626, -0.763924, 1.570796, 2.185761],accel_mss,speed_ms,0,blend_radius_m)
    movel([0.615960, -1.348577, -2.599119, -0.764692, 1.570796, 2.186756],accel_mss,speed_ms,0,blend_radius_m)
    movel([0.617621, -1.344034, -2.602097, -0.766258, 1.570796, 2.188418],accel_mss,speed_ms,0,blend_radius_m)
    movel([0.618283, -1.341640, -2.603655, -0.767094, 1.570796, 2.189079],accel_mss,speed_ms,0,blend_radius_m)
    movel([0.618783, -1.339267, -2.605192, -0.767930, 1.570796, 2.189579],accel_mss,speed_ms,0,blend_radius_m)
    movel([0.619114, -1.336932, -2.606696, -0.768761, 1.570796, 2.189910],accel_mss,speed_ms,0,blend_radius_m)
    movel([0.619273, -1.334640, -2.608165, -0.769584, 1.570796, 2.190069],accel_mss,speed_ms,0,blend_radius_m)
    movel([0.619253, -1.332407, -2.609590, -0.770392, 1.570796, 2.190050],accel_mss,speed_ms,0,blend_radius_m)
    movel([0.619056, -1.330244, -2.610963, -0.771182, 1.570796, 2.189852],accel_mss,speed_ms,0,blend_radius_m)
    movel([0.618673, -1.328162, -2.612279, -0.771948, 1.570796, 2.189470],accel_mss,speed_ms,0,blend_radius_m)
    speed_ms = 0.005
    movel([0.618673, -1.318990, -2.608056, -0.785343, 1.570796, 2.189470],accel_mss,speed_ms,0,blend_radius_m)
    speed_ms = 0.040
    movel([0.608287, -1.336883, -2.596709, -0.778797, 1.570796, 2.179083],accel_mss,speed_ms,0,blend_radius_m)
    speed_ms = 0.005
    movel([0.608287, -1.345938, -2.600853, -0.765598, 1.570796, 2.179083],accel_mss,speed_ms,0,blend_radius_m)
    speed_ms = 0.025
    movel([0.607618, -1.343589, -2.602388, -0.766412, 1.570796, 2.178415],accel_mss,speed_ms,0,blend_radius_m)
    movel([0.606621, -1.341427, -2.603794, -0.767169, 1.570796, 2.177417],accel_mss,speed_ms,0,blend_radius_m)
    movel([0.605939, -1.340487, -2.604403, -0.767499, 1.570796, 2.176735],accel_mss,speed_ms,0,blend_radius_m)
    movel([0.605103, -1.339682, -2.604923, -0.767783, 1.570796, 2.175900],accel_mss,speed_ms,0,blend_radius_m)
    movel([0.604092, -1.339042, -2.605337, -0.768010, 1.570796, 2.174888],accel_mss,speed_ms,0,blend_radius_m)
    movel([0.602882, -1.338593, -2.605627, -0.768169, 1.570796, 2.173679],accel_mss,speed_ms,0,blend_radius_m)
    speed_ms = 0.005
    movel([0.602882, -1.329489, -2.601450, -0.781450, 1.570796, 2.173679],accel_mss,speed_ms,0,blend_radius_m)
    speed_ms = 0.040
    movel([0.608939, -1.326488, -2.603353, -0.782548, 1.570796, 2.179736],accel_mss,speed_ms,0,blend_radius_m)
    speed_ms = 0.005
    movel([0.608939, -1.335612, -2.607543, -0.769234, 1.570796, 2.179736],accel_mss,speed_ms,0,blend_radius_m)
    speed_ms = 0.025
    movel([0.610243, -1.333197, -2.609086, -0.770105, 1.570796, 2.181039],accel_mss,speed_ms,0,blend_radius_m)
    movel([0.611107, -1.330823, -2.610596, -0.770970, 1.570796, 2.181903],accel_mss,speed_ms,0,blend_radius_m)
    movel([0.611540, -1.328533, -2.612045, -0.771811, 1.570796, 2.182336],accel_mss,speed_ms,0,blend_radius_m)
    movel([0.611538, -1.326385, -2.613398, -0.772606, 1.570796, 2.182334],accel_mss,speed_ms,0,blend_radius_m)
    movel([0.611105, -1.324430, -2.614624, -0.773336, 1.570796, 2.181902],accel_mss,speed_ms,0,blend_radius_m)
    movel([0.610245, -1.322725, -2.615688, -0.773976, 1.570796, 2.181041],accel_mss,speed_ms,0,blend_radius_m)
    movel([0.608961, -1.321322, -2.616562, -0.774506, 1.570796, 2.179757],accel_mss,speed_ms,0,blend_radius_m)
    movel([0.608159, -1.320752, -2.616916, -0.774722, 1.570796, 2.178955],accel_mss,speed_ms,0,blend_radius_m)
    movel([0.607255, -1.320275, -2.617211, -0.774903, 1.570796, 2.178051],accel_mss,speed_ms,0,blend_radius_m)
    speed_ms = 0.005
    movel([0.607255, -1.311053, -2.612952, -0.788384, 1.570796, 2.178051],accel_mss,speed_ms,0,blend_radius_m)
    speed_ms = 0.040
    movel([0.613864, -1.309274, -2.614039, -0.789077, 1.570796, 2.184660],accel_mss,speed_ms,0,blend_radius_m)
    speed_ms = 0.005
    movel([0.613864, -1.318507, -2.618305, -0.775576, 1.570796, 2.184660],accel_mss,speed_ms,0,blend_radius_m)
    speed_ms = 0.025
    movel([0.614362, -1.317270, -2.619068, -0.776050, 1.570796, 2.185158],accel_mss,speed_ms,0,blend_radius_m)
    movel([0.614733, -1.316020, -2.619838, -0.776531, 1.570796, 2.185530],accel_mss,speed_ms,0,blend_radius_m)
    movel([0.615108, -1.313519, -2.621370, -0.777500, 1.570796, 2.185904],accel_mss,speed_ms,0,blend_radius_m)
    movel([0.615013, -1.311091, -2.622850, -0.778448, 1.570796, 2.185809],accel_mss,speed_ms,0,blend_radius_m)
    movel([0.614473, -1.308828, -2.624222, -0.779339, 1.570796, 2.185269],accel_mss,speed_ms,0,blend_radius_m)
    movel([0.613517, -1.306811, -2.625439, -0.780138, 1.570796, 2.184314],accel_mss,speed_ms,0,blend_radius_m)
    movel([0.612179, -1.305135, -2.626447, -0.780807, 1.570796, 2.182975],accel_mss,speed_ms,0,blend_radius_m)
    movel([0.611372, -1.304453, -2.626856, -0.781080, 1.570796, 2.182168],accel_mss,speed_ms,0,blend_radius_m)
    movel([0.609512, -1.303452, -2.627455, -0.781482, 1.570796, 2.180308],accel_mss,speed_ms,0,blend_radius_m)
    movel([0.608466, -1.303155, -2.627633, -0.781601, 1.570796, 2.179262],accel_mss,speed_ms,0,blend_radius_m)
    speed_ms = 0.005
    movel([0.608466, -1.293828, -2.623296, -0.795265, 1.570796, 2.179262],accel_mss,speed_ms,0,blend_radius_m)
    speed_ms = 0.040
    movel([0.617198, -1.292574, -2.624034, -0.795781, 1.570796, 2.187994],accel_mss,speed_ms,0,blend_radius_m)
    speed_ms = 0.005
    movel([0.617198, -1.301908, -2.628377, -0.782104, 1.570796, 2.187994],accel_mss,speed_ms,0,blend_radius_m)
    speed_ms = 0.025
    movel([0.617312, -1.299065, -2.630065, -0.783259, 1.570796, 2.188108],accel_mss,speed_ms,0,blend_radius_m)
    movel([0.617008, -1.296386, -2.631647, -0.784356, 1.570796, 2.187804],accel_mss,speed_ms,0,blend_radius_m)
    movel([0.616278, -1.293946, -2.633079, -0.785363, 1.570796, 2.187075],accel_mss,speed_ms,0,blend_radius_m)
    movel([0.615115, -1.291804, -2.634331, -0.786254, 1.570796, 2.185912],accel_mss,speed_ms,0,blend_radius_m)
    movel([0.613512, -1.290032, -2.635361, -0.786996, 1.570796, 2.184309],accel_mss,speed_ms,0,blend_radius_m)
    movel([0.612545, -1.289304, -2.635784, -0.787301, 1.570796, 2.183341],accel_mss,speed_ms,0,blend_radius_m)
    movel([0.611467, -1.288695, -2.636136, -0.787558, 1.570796, 2.182263],accel_mss,speed_ms,0,blend_radius_m)
    movel([0.610275, -1.288211, -2.636417, -0.787762, 1.570796, 2.181072],accel_mss,speed_ms,0,blend_radius_m)
    movel([0.608969, -1.287860, -2.636619, -0.787910, 1.570796, 2.179766],accel_mss,speed_ms,0,blend_radius_m)
    movel([0.607554, -1.287651, -2.636740, -0.787998, 1.570796, 2.178350],accel_mss,speed_ms,0,blend_radius_m)
    movel([0.606026, -1.287590, -2.636775, -0.788024, 1.570796, 2.176822],accel_mss,speed_ms,0,blend_radius_m)
    speed_ms = 0.005
    movel([0.606026, -1.278173, -2.632367, -0.801848, 1.570796, 2.176822],accel_mss,speed_ms,0,blend_radius_m)
    speed_ms = 0.040
    movel([0.616189, -1.275408, -2.633938, -0.803043, 1.570796, 2.186985],accel_mss,speed_ms,0,blend_radius_m)
    speed_ms = 0.005
    movel([0.616189, -1.284841, -2.638358, -0.789190, 1.570796, 2.186985],accel_mss,speed_ms,0,blend_radius_m)
    speed_ms = 0.025
    movel([0.616786, -1.282923, -2.639456, -0.790010, 1.570796, 2.187583],accel_mss,speed_ms,0,blend_radius_m)
    movel([0.617111, -1.281060, -2.640519, -0.790811, 1.570796, 2.187908],accel_mss,speed_ms,0,blend_radius_m)
    movel([0.617157, -1.279285, -2.641527, -0.791577, 1.570796, 2.187953],accel_mss,speed_ms,0,blend_radius_m)
    movel([0.616917, -1.277640, -2.642458, -0.792292, 1.570796, 2.187714],accel_mss,speed_ms,0,blend_radius_m)
    movel([0.616271, -1.275858, -2.643462, -0.793069, 1.570796, 2.187067],accel_mss,speed_ms,0,blend_radius_m)
    movel([0.615324, -1.274279, -2.644349, -0.793761, 1.570796, 2.186120],accel_mss,speed_ms,0,blend_radius_m)
    movel([0.613936, -1.272635, -2.645269, -0.794486, 1.570796, 2.184732],accel_mss,speed_ms,0,blend_radius_m)
    movel([0.612259, -1.271257, -2.646037, -0.795095, 1.570796, 2.183056],accel_mss,speed_ms,0,blend_radius_m)
    movel([0.610290, -1.270206, -2.646622, -0.795562, 1.570796, 2.181086],accel_mss,speed_ms,0,blend_radius_m)
    movel([0.608020, -1.269545, -2.646989, -0.795856, 1.570796, 2.178817],accel_mss,speed_ms,0,blend_radius_m)
    movel([0.605453, -1.269343, -2.647101, -0.795946, 1.570796, 2.176250],accel_mss,speed_ms,0,blend_radius_m)
    movel([0.604079, -1.269427, -2.647054, -0.795908, 1.570796, 2.174875],accel_mss,speed_ms,0,blend_radius_m)
    movel([0.601207, -1.269986, -2.646744, -0.795659, 1.570796, 2.172003],accel_mss,speed_ms,0,blend_radius_m)
    movel([0.599734, -1.270459, -2.646481, -0.795449, 1.570796, 2.170531],accel_mss,speed_ms,0,blend_radius_m)
    movel([0.598254, -1.271070, -2.646141, -0.795178, 1.570796, 2.169050],accel_mss,speed_ms,0,blend_radius_m)
    movel([0.596777, -1.271817, -2.645725, -0.794847, 1.570796, 2.167573],accel_mss,speed_ms,0,blend_radius_m)
    speed_ms = 0.005
    movel([0.596777, -1.262313, -2.641245, -0.808830, 1.570796, 2.167573],accel_mss,speed_ms,0,blend_radius_m)
    speed_ms = 0.040
    movel([0.610162, -1.255273, -2.645088, -0.812028, 1.570796, 2.180958],accel_mss,speed_ms,0,blend_radius_m)
    speed_ms = 0.005
    movel([0.610162, -1.264814, -2.649599, -0.797976, 1.570796, 2.180958],accel_mss,speed_ms,0,blend_radius_m)
    speed_ms = 0.025
    movel([0.608223, -1.262806, -2.650699, -0.798885, 1.570796, 2.179019],accel_mss,speed_ms,0,blend_radius_m)
    movel([0.605896, -1.261103, -2.651627, -0.799658, 1.570796, 2.176692],accel_mss,speed_ms,0,blend_radius_m)
    movel([0.603204, -1.259803, -2.652334, -0.800252, 1.570796, 2.174000],accel_mss,speed_ms,0,blend_radius_m)
    movel([0.601731, -1.259331, -2.652590, -0.800468, 1.570796, 2.172527],accel_mss,speed_ms,0,blend_radius_m)
    movel([0.600177, -1.258994, -2.652773, -0.800622, 1.570796, 2.170973],accel_mss,speed_ms,0,blend_radius_m)
    movel([0.598548, -1.258803, -2.652876, -0.800710, 1.570796, 2.169344],accel_mss,speed_ms,0,blend_radius_m)
    movel([0.596850, -1.258769, -2.652894, -0.800725, 1.570796, 2.167646],accel_mss,speed_ms,0,blend_radius_m)
    movel([0.595084, -1.258904, -2.652822, -0.800664, 1.570796, 2.165881],accel_mss,speed_ms,0,blend_radius_m)
    movel([0.593255, -1.259219, -2.652651, -0.800519, 1.570796, 2.164052],accel_mss,speed_ms,0,blend_radius_m)
    movel([0.591368, -1.259721, -2.652378, -0.800289, 1.570796, 2.162164],accel_mss,speed_ms,0,blend_radius_m)
    movel([0.589429, -1.260425, -2.651996, -0.799968, 1.570796, 2.160226],accel_mss,speed_ms,0,blend_radius_m)
    movel([0.587443, -1.261337, -2.651500, -0.799552, 1.570796, 2.158239],accel_mss,speed_ms,0,blend_radius_m)
    movel([0.585414, -1.262471, -2.650882, -0.799036, 1.570796, 2.156210],accel_mss,speed_ms,0,blend_radius_m)
    speed_ms = 0.005
    movel([0.585414, -1.252918, -2.646359, -0.813111, 1.570796, 2.156210],accel_mss,speed_ms,0,blend_radius_m)
    speed_ms = 0.040
    movel([0.598369, -1.242369, -2.651976, -0.818045, 1.570796, 2.169165],accel_mss,speed_ms,0,blend_radius_m)
    speed_ms = 0.005
    movel([0.598369, -1.251973, -2.656546, -0.803869, 1.570796, 2.169165],accel_mss,speed_ms,0,blend_radius_m)
    speed_ms = 0.025
    movel([0.597272, -1.251063, -2.657031, -0.804295, 1.570796, 2.168068],accel_mss,speed_ms,0,blend_radius_m)
    movel([0.596023, -1.250312, -2.657430, -0.804646, 1.570796, 2.166820],accel_mss,speed_ms,0,blend_radius_m)
    movel([0.594635, -1.249734, -2.657737, -0.804918, 1.570796, 2.165431],accel_mss,speed_ms,0,blend_radius_m)
    movel([0.593122, -1.249325, -2.657954, -0.805110, 1.570796, 2.163918],accel_mss,speed_ms,0,blend_radius_m)
    movel([0.591496, -1.249090, -2.658079, -0.805220, 1.570796, 2.162292],accel_mss,speed_ms,0,blend_radius_m)
    movel([0.589773, -1.249035, -2.658108, -0.805246, 1.570796, 2.160569],accel_mss,speed_ms,0,blend_radius_m)
    movel([0.587971, -1.249158, -2.658042, -0.805188, 1.570796, 2.158767],accel_mss,speed_ms,0,blend_radius_m)
    movel([0.586097, -1.249465, -2.657880, -0.805044, 1.570796, 2.156894],accel_mss,speed_ms,0,blend_radius_m)
    movel([0.584175, -1.249956, -2.657620, -0.804814, 1.570796, 2.154971],accel_mss,speed_ms,0,blend_radius_m)
    movel([0.582222, -1.250621, -2.657266, -0.804502, 1.570796, 2.153019],accel_mss,speed_ms,0,blend_radius_m)
    movel([0.580260, -1.251450, -2.656825, -0.804114, 1.570796, 2.151056],accel_mss,speed_ms,0,blend_radius_m)
    movel([0.578304, -1.252435, -2.656300, -0.803654, 1.570796, 2.149100],accel_mss,speed_ms,0,blend_radius_m)
    movel([0.576372, -1.253561, -2.655698, -0.803130, 1.570796, 2.147169],accel_mss,speed_ms,0,blend_radius_m)
    movel([0.574480, -1.254823, -2.655022, -0.802544, 1.570796, 2.145277],accel_mss,speed_ms,0,blend_radius_m)
    movel([0.572653, -1.256207, -2.654278, -0.801904, 1.570796, 2.143449],accel_mss,speed_ms,0,blend_radius_m)
    movel([0.570903, -1.257701, -2.653472, -0.801216, 1.570796, 2.141699],accel_mss,speed_ms,0,blend_radius_m)
    speed_ms = 0.005
    movel([0.570903, -1.248125, -2.648928, -0.815336, 1.570796, 2.141699],accel_mss,speed_ms,0,blend_radius_m)
    speed_ms = 0.040
    movel([0.581833, -1.236261, -2.655167, -0.820961, 1.570796, 2.152630],accel_mss,speed_ms,0,blend_radius_m)
    speed_ms = 0.005
    movel([0.581833, -1.245895, -2.659765, -0.806729, 1.570796, 2.152630],accel_mss,speed_ms,0,blend_radius_m)
    speed_ms = 0.025
    movel([0.580655, -1.245118, -2.660174, -0.807098, 1.570796, 2.151451],accel_mss,speed_ms,0,blend_radius_m)
    movel([0.579245, -1.244644, -2.660422, -0.807323, 1.570796, 2.150042],accel_mss,speed_ms,0,blend_radius_m)
    movel([0.577646, -1.244456, -2.660521, -0.807412, 1.570796, 2.148442],accel_mss,speed_ms,0,blend_radius_m)
    movel([0.575895, -1.244521, -2.660487, -0.807381, 1.570796, 2.146691],accel_mss,speed_ms,0,blend_radius_m)
    movel([0.574029, -1.244817, -2.660332, -0.807240, 1.570796, 2.144826],accel_mss,speed_ms,0,blend_radius_m)
    movel([0.572093, -1.245317, -2.660069, -0.807003, 1.570796, 2.142889],accel_mss,speed_ms,0,blend_radius_m)
    movel([0.570122, -1.245989, -2.659716, -0.806684, 1.570796, 2.140919],accel_mss,speed_ms,0,blend_radius_m)
    movel([0.568160, -1.246811, -2.659283, -0.806295, 1.570796, 2.138956],accel_mss,speed_ms,0,blend_radius_m)
    movel([0.566149, -1.247795, -2.658764, -0.805830, 1.570796, 2.136945],accel_mss,speed_ms,0,blend_radius_m)
    movel([0.564149, -1.248921, -2.658168, -0.805300, 1.570796, 2.134946],accel_mss,speed_ms,0,blend_radius_m)
    movel([0.562186, -1.250182, -2.657499, -0.804707, 1.570796, 2.132982],accel_mss,speed_ms,0,blend_radius_m)
    movel([0.560295, -1.251575, -2.656759, -0.804056, 1.570796, 2.131091],accel_mss,speed_ms,0,blend_radius_m)
    movel([0.558508, -1.253085, -2.655953, -0.803352, 1.570796, 2.129305],accel_mss,speed_ms,0,blend_radius_m)
    movel([0.556856, -1.254705, -2.655085, -0.802599, 1.570796, 2.127652],accel_mss,speed_ms,0,blend_radius_m)
    movel([0.555373, -1.256431, -2.654157, -0.801801, 1.570796, 2.126169],accel_mss,speed_ms,0,blend_radius_m)
    movel([0.554087, -1.258250, -2.653175, -0.800964, 1.570796, 2.124883],accel_mss,speed_ms,0,blend_radius_m)
    speed_ms = 0.005
    movel([0.554087, -1.248676, -2.648634, -0.815079, 1.570796, 2.124883],accel_mss,speed_ms,0,blend_radius_m)
    speed_ms = 0.040
    movel([0.560669, -1.236787, -2.654894, -0.820708, 1.570796, 2.131465],accel_mss,speed_ms,0,blend_radius_m)
    speed_ms = 0.005
    movel([0.560669, -1.246418, -2.659490, -0.806481, 1.570796, 2.131465],accel_mss,speed_ms,0,blend_radius_m)
    speed_ms = 0.025
    movel([0.558095, -1.246749, -2.659315, -0.806324, 1.570796, 2.128891],accel_mss,speed_ms,0,blend_radius_m)
    movel([0.555260, -1.247449, -2.658946, -0.805994, 1.570796, 2.126057],accel_mss,speed_ms,0,blend_radius_m)
    movel([0.552301, -1.248510, -2.658386, -0.805493, 1.570796, 2.123097],accel_mss,speed_ms,0,blend_radius_m)
    movel([0.549355, -1.249923, -2.657637, -0.804829, 1.570796, 2.120151],accel_mss,speed_ms,0,blend_radius_m)
    movel([0.546557, -1.251678, -2.656704, -0.804007, 1.570796, 2.117353],accel_mss,speed_ms,0,blend_radius_m)
    movel([0.545253, -1.252682, -2.656168, -0.803539, 1.570796, 2.116050],accel_mss,speed_ms,0,blend_radius_m)
    movel([0.544040, -1.253765, -2.655589, -0.803035, 1.570796, 2.114836],accel_mss,speed_ms,0,blend_radius_m)
    movel([0.542928, -1.254931, -2.654964, -0.802494, 1.570796, 2.113724],accel_mss,speed_ms,0,blend_radius_m)
    movel([0.541935, -1.256174, -2.654296, -0.801920, 1.570796, 2.112732],accel_mss,speed_ms,0,blend_radius_m)
    movel([0.541083, -1.257492, -2.653585, -0.801312, 1.570796, 2.111880],accel_mss,speed_ms,0,blend_radius_m)
    movel([0.540381, -1.258889, -2.652830, -0.800671, 1.570796, 2.111177],accel_mss,speed_ms,0,blend_radius_m)
    speed_ms = 0.005
    movel([0.540381, -1.249318, -2.648291, -0.814780, 1.570796, 2.111177],accel_mss,speed_ms,0,blend_radius_m)
    speed_ms = 0.040
    movel([0.539729, -1.243401, -2.651432, -0.817556, 1.570796, 2.110525],accel_mss,speed_ms,0,blend_radius_m)
    speed_ms = 0.005
    movel([0.539729, -1.253001, -2.655998, -0.803391, 1.570796, 2.110525],accel_mss,speed_ms,0,blend_radius_m)
    speed_ms = 0.025
    movel([0.535561, -1.255244, -2.654796, -0.802350, 1.570796, 2.106357],accel_mss,speed_ms,0,blend_radius_m)
    movel([0.533496, -1.256537, -2.654100, -0.801752, 1.570796, 2.104292],accel_mss,speed_ms,0,blend_radius_m)
    movel([0.531501, -1.257950, -2.653338, -0.801101, 1.570796, 2.102298],accel_mss,speed_ms,0,blend_radius_m)
    movel([0.529616, -1.259495, -2.652501, -0.800393, 1.570796, 2.100412],accel_mss,speed_ms,0,blend_radius_m)
    movel([0.527876, -1.261180, -2.651586, -0.799624, 1.570796, 2.098673],accel_mss,speed_ms,0,blend_radius_m)
    movel([0.526329, -1.263009, -2.650587, -0.798792, 1.570796, 2.097126],accel_mss,speed_ms,0,blend_radius_m)
    movel([0.525007, -1.264994, -2.649500, -0.797895, 1.570796, 2.095803],accel_mss,speed_ms,0,blend_radius_m)
    speed_ms = 0.005
    # Splitting Linear movement in 2 (instruction 3386: MoveL 3110)
    movel([0.525007, -1.241553, -2.638115, -0.832721, 1.570796, 2.095803],accel_mss,speed_ms,0,blend_radius_m)
    movel([0.525007, -1.219449, -2.626381, -0.866560, 1.570796, 2.095803],accel_mss,speed_ms,0,blend_radius_m)
    speed_ms = 1.000
    movel([0.525007, -1.219449, -2.626381, -0.866560, 1.570796, 2.095803],accel_mss,speed_ms,0,blend_radius_m)
    # Splitting Linear movement in 6 (instruction 3389: MoveL 3112)
    movel([0.525007, -1.185458, -2.606099, -0.920831, 1.570796, 2.095803],accel_mss,speed_ms,0,blend_radius_m)
    movel([0.525007, -1.154843, -2.584985, -0.972561, 1.570796, 2.095803],accel_mss,speed_ms,0,blend_radius_m)
    movel([0.525007, -1.127379, -2.563110, -1.021900, 1.570796, 2.095803],accel_mss,speed_ms,0,blend_radius_m)
    movel([0.525007, -1.102846, -2.540541, -1.069003, 1.570796, 2.095803],accel_mss,speed_ms,0,blend_radius_m)
    movel([0.525007, -1.081028, -2.517332, -1.114030, 1.570796, 2.095803],accel_mss,speed_ms,0,blend_radius_m)
    movel([0.525007, -1.061721, -2.493532, -1.157137, 1.570796, 2.095803],accel_mss,speed_ms,0,blend_radius_m)
    # End of main program
  end

  Machining4()
end
